// TIA Portal V20 export
FUNCTION_BLOCK "FB_GestionGripper"   // FB43, SCL
{ S7_Optimized_Access := 'TRUE' }
// stored: MemoryReserve 100, SetENOAutomatically false
   VAR
      sLoadGripperCloseReq : Bool;
      sUnloadGripperCloseReq : Bool;
      sLoadShift : Bool;
      sUnLoadShift : Bool;
      sLoadPartLost : Bool;
      sUnLoadPartLost : Bool;
      sLoadClose : Bool;
      sUnLoadClose : Bool;
      sUndrilledGripper : "FB_Gripper";
      sDrilledGripper : "FB_Gripper";
      sLoadCloseWithPart : Bool;
      sUnLoadCloseWithPart : Bool;
      sLoadOpen : Bool;
      sUnLoadOpen : Bool;
      sFT_ModeJog : F_TRIG;
      sBlowingTimerCmdHMI : TP_TIME;
      sRT_BlowingCmdHMI { S7_SetPoint := 'True'} : R_TRIG;
      sBlowingISO { S7_SetPoint := 'True'} : Bool;
      sGripperStatus : Struct
         Available : Bool;
         DrivedByShuttle1 : Bool;
         DrivedByShuttle2 : Bool;
         DrivedByFixture : Bool;
      END_STRUCT;
      sGripperReq : Struct
         ByShuttle1 : Bool;
         ByShuttle2 : Bool;
         ByFixture : Bool;
      END_STRUCT;
      sUndrilledGripperErrorCode : Int;
      sDrilledGripperErrorCode : Int;
   END_VAR
   VAR_TEMP
      tLoadInCycle : Bool;
      tUnloadInCycle : Bool;
   END_VAR
BEGIN
   REGION Description header 
       //==================================================================================
       // POSALUX Swiss SA / (C) Copyright 2025
       //----------------------------------------------------------------------------------
       // Title: 
       // Comment/Function: 
       // Author: Fabien WALDT
       // Engineering: TIA Portal v17
       //----------------------------------------------------------------------------------
       // Change log table:
       // Version  | Date     | Expert in charge | Changes applied
       // ---------|----------|------------------|-----------------------------------------
       // 00.00.01 | 20250506 | WFA              | First released version
       // =================================================================================
   END_REGION

   REGION Key[4] and Key[5] Management
       // Key[4] : Activating of loading/unloading undrilled part
       // Key[5] : Activation of loading/unloading drilled part

       // Key[4] and Key[5] enabled in Jog Mode
       "DB_McpKeyboardSignals".sK4_GripperUndrilledPart.sKeyDisable := NOT "LBP_ModeGroup".E_JOG OR "DB_GestionWorkingModes".sMCP_KxxKeysDisable;
       "DB_HmiKeyboardSignals".sK4a_GripperUndrilledPartClose.sKeyDisable := NOT "LBP_ModeGroup".E_JOG;
       "DB_HmiKeyboardSignals".sK4b_GripperUndrilledPartOpen.sKeyDisable := NOT "LBP_ModeGroup".E_JOG;
       "DB_McpKeyboardSignals".sK5_GripperDrilledPart.sKeyDisable   := NOT "LBP_ModeGroup".E_JOG OR "DB_GestionWorkingModes".sMCP_KxxKeysDisable;
       "DB_HmiKeyboardSignals".sK5a_GripperDrilledPartClose.sKeyDisable   := NOT "LBP_ModeGroup".E_JOG;
   END_REGION

   REGION Load Gripper Command (Undrilled Part)
       // Load Gripper Close Command
       IF "LBP_Chan1".MDyn[80]     // M80 : Close/vaccum loader load (Undrilled Part)
           OR "DB_LoaderShuttle1".oLoadGripperCloseReq
           OR "DB_LoaderShuttle2".oLoadGripperCloseReq
           OR ("LBP_ModeGroup".E_JOG AND "DB_McpKeyboardSignals".sK4_GripperUndrilledPart.sKeySWTogglePositiveFront) 
           OR ("LBP_ModeGroup".E_JOG AND "DB_HmiKeyboardSignals".sK4a_GripperUndrilledPartClose.sKeySWPositiveFront) THEN
           #sLoadGripperCloseReq := TRUE;
       END_IF;

       // Load Gripper Open Command
        IF "LBP_Chan1".MDyn[81]     // M81 : Open/blowing loader load (Undrilled Part)
            OR "DB_LoaderFixture".oLoadGripperOpenReq
            OR ("LBP_ModeGroup".E_JOG AND "DB_McpKeyboardSignals".sK4_GripperUndrilledPart.sKeySWToggleNegativeFront) 
           OR ("LBP_ModeGroup".E_JOG AND "DB_HmiKeyboardSignals".sK4b_GripperUndrilledPartOpen.sKeySWPositiveFront) THEN
           #sLoadGripperCloseReq := FALSE;
        END_IF;
       "DB_McpKeyboardSignals".sK4_GripperUndrilledPart.sKeySWToggleStatus := #sLoadGripperCloseReq;
      // "DB_HmiKeyboardSignals".sK4a_GripperUndrilledPartClose.sKeySWToggleStatus := #sLoadGripperCloseReq;
   END_REGION

   REGION Unload Gripper Command (Drilled Part)  
       // Unload Gripper Close Command
       IF "LBP_Chan1".MDyn[82]     // M82 : Close/vaccum loader unload (Drilled Part)
           OR "DB_LoaderFixture".oUnloadGripperCloseReq
           OR ("LBP_ModeGroup".E_JOG AND "DB_McpKeyboardSignals".sK5_GripperDrilledPart.sKeySWTogglePositiveFront)
           OR ("LBP_ModeGroup".E_JOG AND "DB_HmiKeyboardSignals".sK5a_GripperDrilledPartClose.sKeySWPositiveFront) THEN
           #sUnloadGripperCloseReq := TRUE;
       END_IF;

       // Unload Gripper Open Command
        IF "LBP_Chan1".MDyn[83]     // M83 : Open/blowing loader unload (Drilled Part)
           // OR #sLoadPartLost
           OR "DB_LoaderShuttle1".oUnloadGripperOpenReq
            OR "DB_LoaderShuttle2".oUnloadGripperOpenReq
         OR ("LBP_ModeGroup".E_JOG AND "DB_McpKeyboardSignals".sK5_GripperDrilledPart.sKeySWToggleNegativeFront)
          OR ("LBP_ModeGroup".E_JOG AND "DB_HmiKeyboardSignals".sK5b_GripperDrilledPartOpen.sKeySWTogglePositiveFront) THEN
            #sUnloadGripperCloseReq := FALSE;
       END_IF;
       "DB_McpKeyboardSignals".sK5_GripperDrilledPart.sKeySWToggleStatus := #sUnloadGripperCloseReq;
       "DB_HmiKeyboardSignals".sK5a_GripperDrilledPartClose.sKeySWToggleStatus := #sUnloadGripperCloseReq;
   END_REGION

   REGION Keys - LED Management
       // KEY - LED [4]: Loading (Undrilled part)
       "DB_McpKeyboardSignals".sK4_GripperUndrilledPart.sKeySWStatus :=
       #sLoadGripperCloseReq
       AND "DB_DecodChannels".sChan1IsDisplayed;

       "DB_HmiKeyboardSignals".sK4a_GripperUndrilledPartClose.sKeySWStatus :=
       #sLoadGripperCloseReq
       AND "DB_DecodChannels".sChan1IsDisplayed;

       "DB_HmiKeyboardSignals".sK4b_GripperUndrilledPartOpen.sKeySWStatus :=
       NOT #sLoadGripperCloseReq
       AND "DB_DecodChannels".sChan1IsDisplayed;

       "DB_McpKeyboardSignals".sK4_GripperUndrilledPart.sLedSWStatus := "DB_McpKeyboardSignals".sK4_GripperUndrilledPart.sKeySWStatus;
       "DB_HmiKeyboardSignals".sK4a_GripperUndrilledPartClose.sLedSWStatus := "DB_HmiKeyboardSignals".sK4a_GripperUndrilledPartClose.sKeySWStatus;
       "DB_HmiKeyboardSignals".sK4b_GripperUndrilledPartOpen.sLedSWStatus := "DB_HmiKeyboardSignals".sK4b_GripperUndrilledPartOpen.sKeySWStatus;

       // KEY - LED [5]: Unloading (Drilled part)
       "DB_McpKeyboardSignals".sK5_GripperDrilledPart.sKeySWStatus :=
       #sUnloadGripperCloseReq
       AND "DB_DecodChannels".sChan1IsDisplayed;

       "DB_HmiKeyboardSignals".sK5a_GripperDrilledPartClose.sKeySWStatus :=
       #sUnloadGripperCloseReq
       AND "DB_DecodChannels".sChan1IsDisplayed;

       "DB_HmiKeyboardSignals".sK5b_GripperDrilledPartOpen.sKeySWStatus :=
       NOT #sUnloadGripperCloseReq
       AND "DB_DecodChannels".sChan1IsDisplayed;

       "DB_McpKeyboardSignals".sK5_GripperDrilledPart.sLedSWStatus := "DB_McpKeyboardSignals".sK5_GripperDrilledPart.sKeySWStatus;
       "DB_HmiKeyboardSignals".sK5a_GripperDrilledPartClose.sLedSWStatus := "DB_HmiKeyboardSignals".sK5a_GripperDrilledPartClose.sKeySWStatus;
       "DB_HmiKeyboardSignals".sK5b_GripperDrilledPartOpen.sLedSWStatus := "DB_HmiKeyboardSignals".sK5b_GripperDrilledPartOpen.sKeySWStatus;
   END_REGION

   REGION Undrilled Gripper        
       #sUndrilledGripper(iHoldPart := #sLoadGripperCloseReq,
                          iOpen := "DB_DigitalInputs".sLoadClampOpened.sSWStatus,
                          iCloseWithoutPart := "DB_DigitalInputs".sLoadClampNotClosedWithPart.sSWStatus,
                          iPulseTime := T#300ms,
                          iMonitorTime:=T#3s,
                          oClose => "DB_DigitalOutputs".sLoadClampClosing.sSWStatus,
                          oOpen => "DB_DigitalOutputs".sLoadClampOpening.sSWStatus,
                          oStateOpen => #sLoadOpen,
                          oStateClose => #sLoadClose,
                          oStateCloseWithPart => #sLoadCloseWithPart,
                          oErrorCode=>#sUndrilledGripperErrorCode);

       "LBP_AlarmMsgs".UserA[08].A70UUxx[14] := #sUndrilledGripperErrorCode = 1;    // Msg: 700814 "Loading Gripper Opening Timeout"
       "LBP_AlarmMsgs".UserA[08].A70UUxx[15] := #sUndrilledGripperErrorCode = 2;    // Msg: 700815 "Loading Gripper Closing Timeout"   
   END_REGION

   REGION Drilled Gripper
       #sDrilledGripper(iHoldPart := #sUnloadGripperCloseReq,
                        iOpen := "DB_DigitalInputs".sUnloadClampOpened.sSWStatus,
                        iCloseWithoutPart := "DB_DigitalInputs".sUnloadClampNotClosedWithPart.sSWStatus,
                        iPulseTime := T#300ms,
                        iMonitorTime:=T#3s,
                        oClose => "DB_DigitalOutputs".sUnloadClampClosing.sSWStatus,
                        oOpen => "DB_DigitalOutputs".sUnloadClampOpening.sSWStatus,
                        oStateOpen => #sUnLoadOpen,
                        oStateClose => #sUnLoadClose,
                        oStateCloseWithPart => #sUnLoadCloseWithPart,
                        oErrorCode=>#sDrilledGripperErrorCode);

       "LBP_AlarmMsgs".UserA[08].A70UUxx[16] := #sUndrilledGripperErrorCode = 1;    // Msg: 700816 "Unloading Gripper Opening Timeout"
       "LBP_AlarmMsgs".UserA[08].A70UUxx[17] := #sUndrilledGripperErrorCode = 2;    // Msg: 700817 "Unloading Gripper Closing Timeout"   
   END_REGION

   REGION Blowing
       // Blowing from ISO Code
       IF "LBP_Chan1".MDyn[96] THEN
           #sBlowingISO := TRUE;
       ELSIF "LBP_Chan1".MDyn[97] OR "LBP_Chan1".A_Reset THEN
           #sBlowingISO := FALSE;
       END_IF;

       #sRT_BlowingCmdHMI(CLK := "DB_HMICmd".BlowingCmd);

       #sBlowingTimerCmdHMI(IN := #sRT_BlowingCmdHMI.Q,
                      PT := REAL_TO_DINT("DB_HMISetting".BlowingSetpoint));

       "DB_DigitalOutputs".sBlowing.sSWStatus := "DB_LoaderShuttle1".oBlowingReq
       OR "DB_LoaderShuttle2".oBlowingReq
       OR "DB_LoaderFixture".oBlowingReq
       OR  #sBlowingTimerCmdHMI.Q;

       "DB_HMICmd".BlowingCmd := FALSE;
   END_REGION

   REGION Gripper Status
       IF "DB_LoaderShuttle1".sMain.oGripperAxisRequest AND #sGripperStatus.Available AND NOT "DB_CommPLC_ISO".sAxisReservedbyNC THEN
           #sGripperStatus.Available := FALSE;
           #sGripperStatus.DrivedByShuttle1 := TRUE;
           #sGripperStatus.DrivedByShuttle2 := FALSE;
           #sGripperStatus.DrivedByFixture := FALSE;
       ELSIF "DB_LoaderShuttle2".sMain.oGripperAxisRequest AND #sGripperStatus.Available  AND NOT "DB_CommPLC_ISO".sAxisReservedbyNC THEN
           #sGripperStatus.Available := FALSE;
           #sGripperStatus.DrivedByShuttle1 := FALSE;
           #sGripperStatus.DrivedByShuttle2 := TRUE;
           #sGripperStatus.DrivedByFixture := FALSE;
       ELSIF #sGripperReq.ByFixture AND #sGripperStatus.Available  AND "DB_CommPLC_ISO".sAxisReservedbyNC THEN
           #sGripperStatus.Available := FALSE;
           #sGripperStatus.DrivedByShuttle1 := FALSE;
           #sGripperStatus.DrivedByShuttle2 := FALSE;
           #sGripperStatus.DrivedByFixture := TRUE;
       END_IF;

       IF "DB_LoaderShuttle1".sMain.oGripperAxisRelease THEN
           #sGripperStatus.DrivedByShuttle1 := FALSE;
       END_IF;
       IF "DB_LoaderShuttle2".sMain.sGripperAxisRelease THEN
           #sGripperStatus.DrivedByShuttle2 := FALSE;
       END_IF;
       IF NOT #sGripperReq.ByFixture THEN
           #sGripperStatus.DrivedByFixture := FALSE;
       END_IF;

       IF NOT #sGripperStatus.DrivedByShuttle1
           AND NOT #sGripperStatus.DrivedByShuttle2
           AND NOT #sGripperStatus.DrivedByFixture THEN
           #sGripperStatus.Available := TRUE;
           #sGripperStatus.DrivedByShuttle1 := FALSE;
           #sGripperStatus.DrivedByShuttle2 := FALSE;
           #sGripperStatus.DrivedByFixture := FALSE;
       END_IF;
   END_REGION
END_FUNCTION_BLOCK
